// TwinCAT 3 PLC project DeviceInfo
// Title: TestZeugwerkCreator_Philipp
// Company: philipp
// Author: Philipp Hagen
// ProjectVersion: 1.0.0.1
// ProgramVersion: 3.1.4026.12
// libraries:
//   Tc2_IoFunctions, 3.4.4.0 (Beckhoff Automation GmbH)
//   Tc2_Standard, * (Beckhoff Automation GmbH)
//   Tc2_System, * (Beckhoff Automation GmbH)
//   Tc2_Utilities, * (Beckhoff Automation GmbH)
//   Tc3_Module, * (Beckhoff Automation GmbH)
//   Testbench, 1.0.0.0 (Zeugwerk GmbH)
// project tree:
//   / fb_test.TcPOU
//   Tests/ fb_testTest.TcPOU

// ---- fb_test.TcPOU
/// this is my first test fb
/// some more doc
FUNCTION_BLOCK fb_test
VAR_INPUT
END_VAR
VAR_OUTPUT
	o_ui_countValue		:UINT;
END_VAR
VAR
END_VAR

METHOD Count : BOOL
VAR_INPUT
	i_ui_countCalue			:uint;
END_VAR
o_ui_countValue:=o_ui_countValue+i_ui_countCalue;
END_METHOD

END_FUNCTION_BLOCK

// ---- Tests/fb_testTest.TcPOU
FUNCTION_BLOCK fb_testTest EXTENDS fb_test IMPLEMENTS Testbench.IUnitTest

METHOD Test_CheckCount
VAR_INPUT
  assertions : Testbench.IAssertions;
END_VAR
VAR CONSTANT
  amsNetId : Tc2_System.T_AmsNetID := '5.5.5.5.1.1';
  deviceId : UDINT := 9;
END_VAR
Count(1);
assertions.EqualsUint(1,SUPER^.o_ui_countValue,'Value not 1');
Count(2);
assertions.EqualsUint(3,SUPER^.o_ui_countValue,'Value not 3');
END_METHOD

END_FUNCTION_BLOCK
